FUNCTION IsValidStatus : BOOL
VAR_INPUT
	Status : I_Content;
END_VAR

IsValidStatus := Status <> 0;

END_FUNCTION

(* stored: Version 1.1.0.1, ProductVersion 3.1.4024.12
   POU IsValidStatus: Id {52289197-8d57-0a07-3a3e-607899a0d302}, SpecialFunc None *)
